// TIA Portal V17 export
// export: Created 2025-03-07T09:19:37.7649402Z, ExportSetting WithDefaults, DisplayName Totally Integrated Automation Portal, DisplayVersion V17 Update 8, DisplayName TIA Portal Openness, DisplayVersion V17 Update 8, DisplayName TIA Portal Version Control Interface, DisplayVersion V17, DisplayName SINAMICS Startdrive Advanced, DisplayVersion V17 SP2, DisplayName SINAMICS Startdrive G110M, G120, G120C, G120D, G120P, G115D, DisplayVersion V17 SP2, DisplayName SINAMICS Startdrive G130, G150, S120, S150, SINAMICS MV, S210, DisplayVersion V17 SP2, DisplayName STEP 7 Professional, DisplayVersion V17 Update 8, DisplayName SINUMERIK ONE STEP 7 Toolbox, DisplayVersion V17 Update 12, DisplayName SINUMERIK 840D sl STEP 7 Toolbox, DisplayVersion V17 Update 12, DisplayName STEP 7 Safety, DisplayVersion V17 Update 6, DisplayName WinCC Advanced, DisplayVersion V17 Update 8
TYPE "LBP_typeNCVariableTokenReal"
TITLE = LBP_ReadVar and LBP_WriteVar Interface / Interfaz LBP_ReadVar y LBP_WriteVar / LBP_ReadVar und LBP_WriteVar Schnittstelle
// User Data Type for LBP_ReadVar[FB2] and LBP_WriteVar[FB3] Parameters / Tipo de datos de usuario para parámetros LBP_ReadVar[FB2] y LBP_WriteVar[FB3] / Anwenderdatentyp für LBP_ReadVar[FB2] und LBP_WriteVar[FB3] Parameter
// stored: IsFailsafeCompliant false
   STRUCT
      token : "LBP_typeNCVariableToken";   // Anwenderdatentyp für LBP_ReadVar[FB2] und LBP_WriteVar[FB3] Eingangsparameter Addrx / User Data Type for LBP_ReadVar[FB2] and LBP_WriteVar[FB3] Input Parameter Addrx / Tipo de datos de usuario para parámetros de entrada Addrx LBP_ReadVar[FB2] y LBP_WriteVar[FB3]
      value : Real;   // Datentyp für LBP_ReadVar[FB2] und LBP_WriteVar[FB3] E/A-Parameter SDx / Data Type for LBP_ReadVar[FB2] and LBP_WriteVar[FB3] InOut Parameter SDx / Tipo de datos para parámetros E/S SDx LBP_ReadVar[FB2] y LBP_WriteVar[FB3]
   END_STRUCT;
END_TYPE
